// TIA Portal V20 export
TYPE "typeCmHmiInterfaceBrakeTest"
// stored: Access Published, Namespace Unit1.Em13
   STRUCT
      jrUnloadingPnPAxisZ : "LER_typeBrakeTestEmInterface";
   END_STRUCT;
END_TYPE
